Fanuc KAREL source: ka00014.KL

-- PROVISIONAL review KL for V940-1; original PC SHA256 47d29f947ca1e7f519bf7891168e69afbebae94fcaa483eeae862d15b6a4c80a
-- Incomplete behavior may be omitted. Consult companion uncertainty JSON. Do not deploy.
PROGRAM KA00014
%NOLOCKGROUP
VAR
  SRC : REAL
  DST : REAL
BEGIN
  -- V9_ZERO_TABLE_METADATA_HINT layout=0001; no indexed target words; source/name/runtime held
  -- UNRESOLVED_PC offsets 5-16; opcodes 2E,23
  -- UNRESOLVED_PC offsets 21-33; opcodes 21,23
  -- UNRESOLVED_PC offsets 38-42; opcodes 7F
END KA00014
